FUNCTION_BLOCK FB_FilterSecondaries
VAR_INPUT
    bExecute : BOOL;
    sMotorProduct : STRING;
    nAddrSize : BYTE;
    aAddr     : POINTER TO UINT;
END_VAR
VAR_OUTPUT
    bBusy : BOOL := FALSE;  
    nNumberFound : BYTE := 0;
END_VAR
VAR_IN_OUT
END_VAR
VAR
    fbGetSecondaryInfo : FB_EcGetSlaveIdentity;

    eState : E_State := E_State.Init;
    nCurrIndex : BYTE := 0;
    nLoopVar : BYTE := 0;
    sCurrStr : STRING;
END_VAR

CASE eState OF
E_State.Init:
;
END_CASE

END_FUNCTION_BLOCK

(* stored: Version 1.1.0.1, ProductVersion 3.1.4022.18
   POU FB_FilterSecondaries: Id {ff01b56a-17ce-43f7-9e9f-a72caca7f8b0}, SpecialFunc None *)
